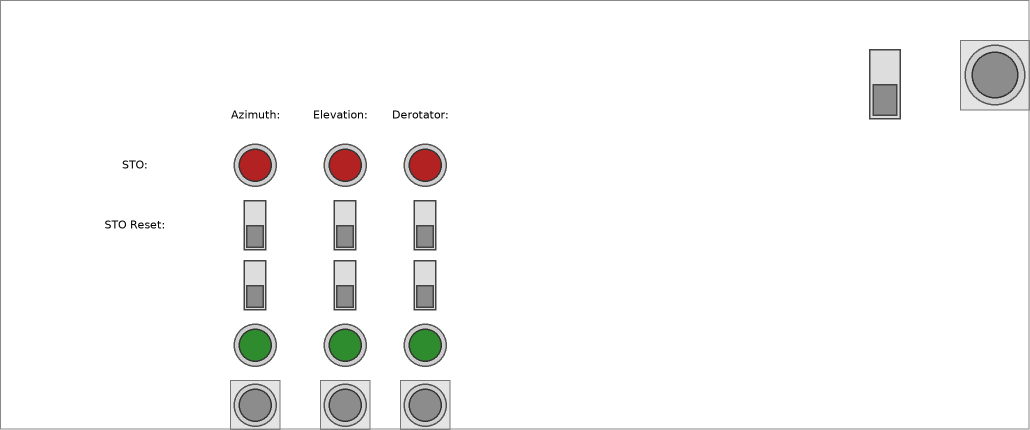
VISUALIZATION STO  // 1030x430
    Label (210,100 91x30), "Azimuth:"
    Lamp1 (230,140 50x50), variable: GVL_Telescope.Azimuth_sto, style: Lamp-Lamp1-Red
    Label (300,100 81x30), "Elevation:"
    Lamp1 (320,140 50x50), variable: GVL_Telescope.Elevation_sto, style: Lamp-Lamp1-Red
    Label (380,100 81x30), "Derotator:"
    Lamp1 (400,140 50x50), variable: GVL_Telescope.Derotator_sto, style: Lamp-Lamp1-Red
    Label (60,150 150x30), "STO:"
    Lamp1 (230,320 50x50), variable: AzimuthElevationControl.ready, style: Lamp-Lamp1-Green
    Lamp1 (320,320 50x50), variable: ElevationControl.Ready, style: Lamp-Lamp1-Green
    Lamp1 (400,320 50x50), style: Lamp-Lamp1-Green
    PushSwitch (230,380 50x50), variable: AzimuthElevationControl.Reset, behaviour: TAP, style: Switch-PushSwitch-Gray
    PushSwitch (320,380 50x50), variable: ElevationControl.reset, behaviour: TAP, style: Switch-PushSwitch-Gray
    PushSwitch (400,380 50x50), behaviour: TAP, style: Switch-PushSwitch-Gray
    DipSwitch (230,260 50x50), variable: AzimuthElevationControl.Enable, behaviour: TOGGLE, style: Switch-DipSwitch-Gray
    DipSwitch (320,260 50x50), variable: ElevationControl.enable, behaviour: TOGGLE, style: Switch-DipSwitch-Gray
    DipSwitch (400,260 50x50), variable: DerotatorControl.enable, behaviour: TOGGLE, style: Switch-DipSwitch-Gray
    DipSwitch (850,49 70x70), variable: GVL_Safety.Restart, behaviour: TOGGLE, style: Switch-DipSwitch-Gray
    PushSwitchLed (960,40 70x70), behaviour: TAP, style: Switch-PushSwitchLed-Gray
    DipSwitch (400,200 50x50), variable: GVL_Safety.Reset_STO_Derotator, behaviour: TOGGLE, style: Switch-DipSwitch-Gray
    DipSwitch (230,200 50x50), variable: GVL_Safety.Reset_STO_Azimuth, behaviour: TOGGLE, style: Switch-DipSwitch-Gray
    DipSwitch (320,200 50x50), variable: GVL_Safety.Reset_STO_Elevation, behaviour: TOGGLE, style: Switch-DipSwitch-Gray
    Label (60,210 150x30), "STO Reset:"
END_VISUALIZATION

(* stored: Version 1.1.0.1, ProductVersion 3.1.4024.12
   Visu STO: Id {2c72abb1-52b7-4434-8d69-25eedaf9331f} *)
